{attribute 'GeneratedUsingTerminal: EL2252--0000'}
{attribute addProperty BoxType "EL2252--0000"}
{attribute addProperty Id "ActivateAT %Q*USINT1"}
{attribute addProperty CRC "4197263632"}
{attribute addProperty Size "1"}
TYPE DC_Sync_Activate_FA2D2910 :
STRUCT
	{attribute addProperty Name "Activate"}
	Activate AT %Q* : USINT;
END_STRUCT
END_TYPE

(* stored: Version 1.2.0.0, ProductVersion 3.1.4024.9
   DUT DC_Sync_Activate_FA2D2910: Id {1ef47aa2-298f-43b3-a90f-4e08e75c6884} *)
